% RSLogix 500 project I2P HANDS-ON 3 - CAYLEN.RSS, saved by version 10.00.00.00 %
PROJECT "ML06B"    % processor: Bul.1763 MicroLogix 1100 Series B %

PROGRAM FILES
  LAD 2   9 rungs

DATA FILES
  O0 OUTPUT  4 elements
  I1 INPUT  6 elements
  S2 STATUS  66 elements
  B3 BINARY  1 elements
  T4 TIMER  1 elements
  C5 COUNTER  1 elements
  R6 CONTROL  1 elements
  N7 INTEGER  1 elements
  F8 FLOAT  1 elements

LADDER 2
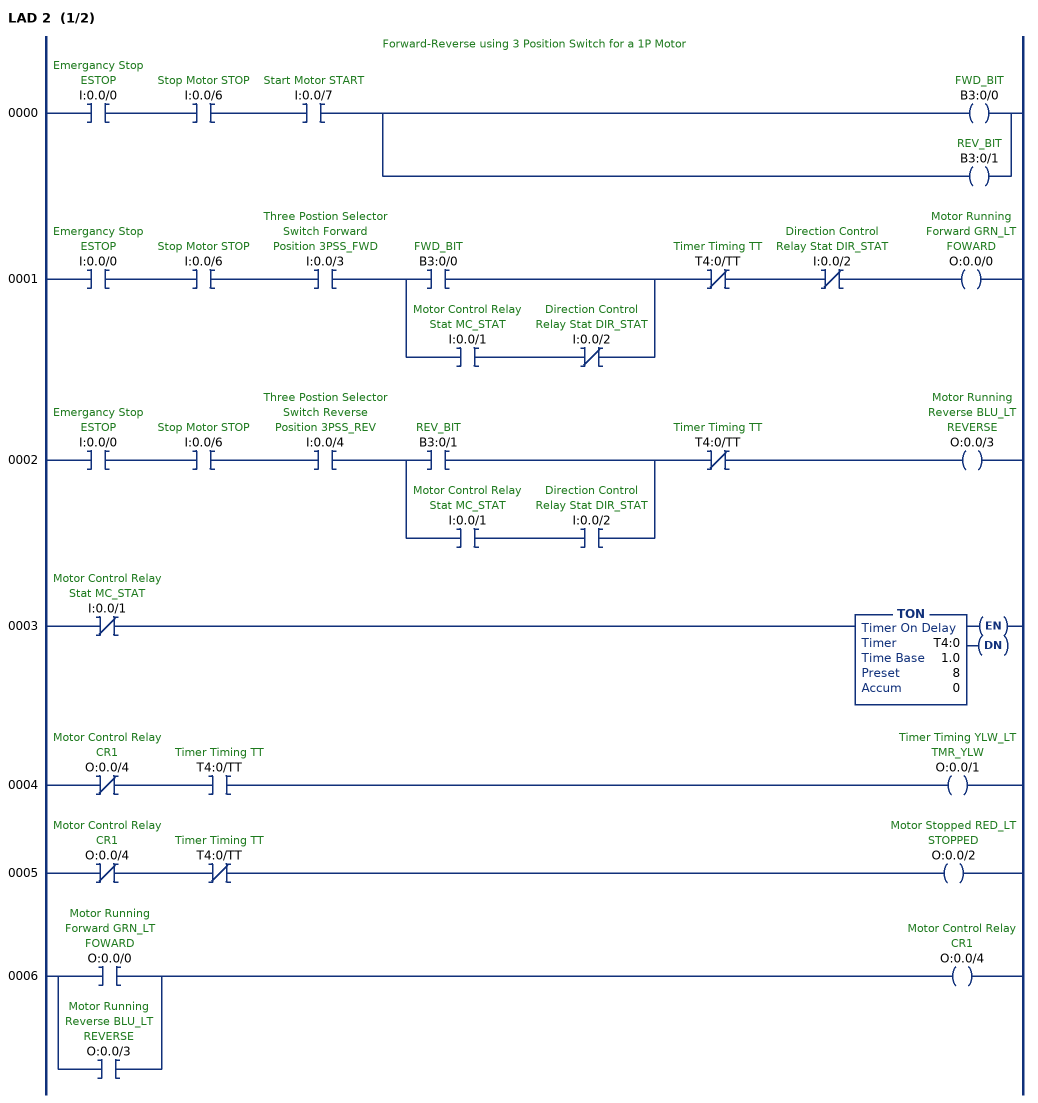
% Rung: 0 %
% Forward-Reverse using 3 Position Switch for a 1P Motor %
SOR XIC I:0.0/0 XIC I:0.0/6 XIC I:0.0/7 BST OTE B3:0/0 NXB OTE B3:0/1 BND EOR
%   I:0.0/0  ESTOP  "Emergancy Stop" %
%   I:0.0/6  STOP  "Stop Motor" %
%   I:0.0/7  START  "Start Motor" %
%   B3:0/0  FWD_BIT %
%   B3:0/1  REV_BIT %
% Rung: 1 %
SOR XIC I:0.0/0 XIC I:0.0/6 XIC I:0.0/3 BST XIC B3:0/0 NXB XIC I:0.0/1 XIO I:0.0/2 BND XIO T4:0/TT XIO I:0.0/2 OTE O:0.0/0 EOR
%   I:0.0/0  ESTOP  "Emergancy Stop" %
%   I:0.0/6  STOP  "Stop Motor" %
%   I:0.0/3  3PSS_FWD  "Three Postion Selector Switch Forward Position" %
%   B3:0/0  FWD_BIT %
%   I:0.0/1  MC_STAT  "Motor Control Relay Stat" %
%   I:0.0/2  DIR_STAT  "Direction Control Relay Stat" %
%   T4:0/TT  TT  "Timer Timing" %
%   O:0.0/0  FOWARD  "Motor Running Forward GRN_LT" %
% Rung: 2 %
SOR XIC I:0.0/0 XIC I:0.0/6 XIC I:0.0/4 BST XIC B3:0/1 NXB XIC I:0.0/1 XIC I:0.0/2 BND XIO T4:0/TT OTE O:0.0/3 EOR
%   I:0.0/0  ESTOP  "Emergancy Stop" %
%   I:0.0/6  STOP  "Stop Motor" %
%   I:0.0/4  3PSS_REV  "Three Postion Selector Switch Reverse Position" %
%   B3:0/1  REV_BIT %
%   I:0.0/1  MC_STAT  "Motor Control Relay Stat" %
%   I:0.0/2  DIR_STAT  "Direction Control Relay Stat" %
%   T4:0/TT  TT  "Timer Timing" %
%   O:0.0/3  REVERSE  "Motor Running Reverse BLU_LT" %
% Rung: 3 %
SOR XIO I:0.0/1 TON T4:0 1.0 8 0 EOR
%   I:0.0/1  MC_STAT  "Motor Control Relay Stat" %
% Rung: 4 %
SOR XIO O:0.0/4 XIC T4:0/TT OTE O:0.0/1 EOR
%   O:0.0/4  CR1  "Motor Control Relay" %
%   T4:0/TT  TT  "Timer Timing" %
%   O:0.0/1  TMR_YLW  "Timer Timing YLW_LT" %
% Rung: 5 %
SOR XIO O:0.0/4 XIO T4:0/TT OTE O:0.0/2 EOR
%   O:0.0/4  CR1  "Motor Control Relay" %
%   T4:0/TT  TT  "Timer Timing" %
%   O:0.0/2  STOPPED  "Motor Stopped RED_LT" %
% Rung: 6 %
SOR BST XIC O:0.0/0 NXB XIC O:0.0/3 BND OTE O:0.0/4 EOR
%   O:0.0/0  FOWARD  "Motor Running Forward GRN_LT" %
%   O:0.0/3  REVERSE  "Motor Running Reverse BLU_LT" %
%   O:0.0/4  CR1  "Motor Control Relay" %

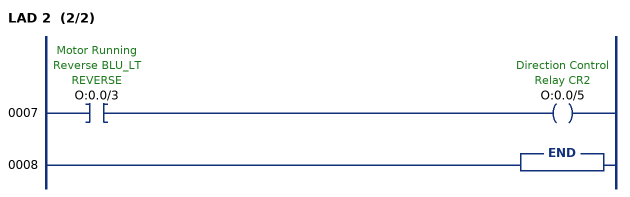
% Rung: 7 %
SOR XIC O:0.0/3 OTE O:0.0/5 EOR
%   O:0.0/3  REVERSE  "Motor Running Reverse BLU_LT" %
%   O:0.0/5  CR2  "Direction Control Relay" %
% Rung: 8 %
SOR END EOR

DATA TABLE (non-zero values as saved)
DATA B3
% B3:0 % 0X0001
DATA T4
% .PRE .ACC %
% T4:0 % 8 0
